FUNCTION_BLOCK Watchdog
VAR_INPUT
	enable : BOOL := TRUE; //watchdog can be disabled if needed
	
	toggleBit : BOOL;
	timeoutWidth : TIME := DEFAULT_ADS_TIMEOUT;
END_VAR
VAR_OUTPUT
	timeout : BOOL;
	prevMsgTimestamp : TIMESTRUCT;
END_VAR
VAR	
	timer : TON;
	memoryBit : BOOL;
END_VAR

timer(
	IN:= enable AND (memoryBit = toggleBit), 
	PT:= timeoutWidth, 
	Q=> timeout, 
	ET=> );
	
IF enable AND memoryBit <> toggleBit THEN
	prevMsgTimestamp := MAIN.localTime;
END_IF

memoryBit := toggleBit;

END_FUNCTION_BLOCK

(* stored: Version 1.1.0.1, ProductVersion 3.1.4024.11
   POU Watchdog: Id {5441069f-d199-4420-9a7a-e035c7bf04a5}, SpecialFunc None *)
